PROGRAM MAIN
VAR
	(* bsp. Timeraufruf Häufigkeit *)
	bTimerIn_call 		: BOOL;
	timer_call_1		: TON;
	timer_call_2		: TON;
	
	iTotalPLCCycles		: INT;
	iCycles 			: INT 		:= 100; // Häufigkeit der timer aufrufe
	iCycles_cnt 		: INT 		:= 100; 	
	iCycles_stop1 		: INT;
	iCycles_stop2 		: INT;
	
	bstop 				: BOOL;
END_VAR


iTotalPLCCycles := iTotalPLCCycles+1;
(* Timer Aufruf *) 

(* timer calls *)
// timer_call_1 wird jeden Zyklus aufgerufen (Neuberechnung von Q und ET erfolgt jeden Zyklus (alle 10 ms))
// timer_call_2 wird jeden 100. Zyklus aufgerufen (Neuberechung von Q und ET erfolgt nur jede Sekunde einmal)
// Fazit: Timer zählt intern weiter. Auflösung der internen Berechnung ist abhängig von der Aufruffrequenz.
iCycles_cnt := iCycles_cnt + 1;
timer_call_1(IN := bTimerIn_call, PT := T#20.1S);



// Reset counter
IF iCycles_cnt >= iCycles THEN
	timer_call_2(IN := bTimerIn_call, PT := T#20.1S);
	iCycles_cnt := 0; // Reset counter
END_IF



// check timer value after 8.3 s
IF timer_call_1.ET = T#8.3S THEN
	bstop := TRUE; 
END_IF

IF timer_call_1.Q THEN
	iCycles_stop1 := iTotalPLCCycles;	
	timer_call_1(IN:= FALSE);
END_IF

IF timer_call_2.Q THEN
	iCycles_stop2 := iTotalPLCCycles;	
	timer_call_2(IN:= FALSE);
END_IF

END_PROGRAM

(* stored: Version 1.1.0.1, ProductVersion 3.1.4024.9
   POU MAIN: Id {5409316e-79f4-408c-a491-4c9c321f4cbd}, SpecialFunc None *)
